PROGRAM Datalogger
VAR_IN_OUT CONSTANT
	monitoring			: ST_System_Monitor;
END_VAR

VAR
	FB_Datalogger					:FB_Datalogger;
END_VAR
VAR CONSTANT
	MAXLREALTOSTRINGLENGTH			: UDINT := 30;	
	NUMBEROFCOLUMNS					: UDINT := 40;													// Total number of columns
	TOTALNUMBEROFROWS				: UDINT := 86400;										    	// Total number of rows in one file (Depends of logtime)
	INCREOFROWS						: UDINT := 5;													// Amount of rows to write at once
	BUFFERMEM						: UDINT := 150;													// Effects file size
	NUMBEROFELEMENTS				: UDINT := NUMBEROFCOLUMNS * INCREOFROWS;						// > NUMBEROFCOLUMNS * INCREOFROWS
	MARGEDATAUSAGE					: REAL  := 0.05;												// 5% Standard marge (95% of storage gets used)
END_VAR
VAR PERSISTENT
	//Datalog presis 
	udi_MaxAmoutOfFiles									: UDINT;								// Max amount of files (30Mb = 12000 ROWS = 10min log)
	udi_AmountOfFiles									: UDINT;
	b_FileNotClosed										: BOOL;
	ui_FileNotClosed									: UINT; 
	a_LogFilesCreated									: ARRAY [0..10000] OF STRING(30);
END_VAR

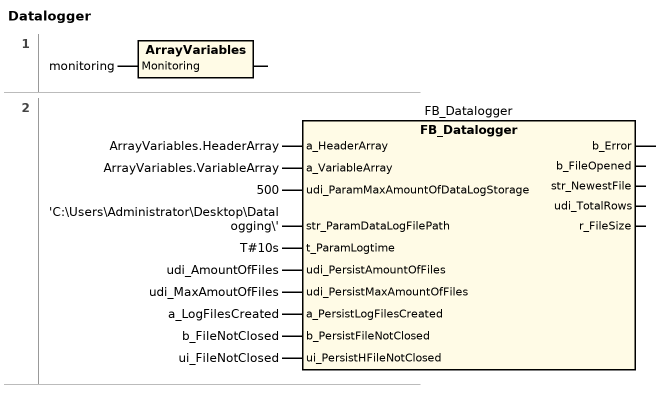
// NETWORK 1
ArrayVariables(Monitoring := monitoring);

// NETWORK 2
FB_Datalogger(
    a_HeaderArray := ArrayVariables.HeaderArray,
    a_VariableArray := ArrayVariables.VariableArray,
    udi_ParamMaxAmountOfDataLogStorage := 500,
    str_ParamDataLogFilePath := 'C:\Users\Administrator\Desktop\Datalogging\',
    t_ParamLogtime := T#10s,
    udi_PersistAmountOfFiles := udi_AmountOfFiles,
    udi_PersistMaxAmountOfFiles := udi_MaxAmoutOfFiles,
    a_PersistLogFilesCreated := a_LogFilesCreated,
    b_PersistFileNotClosed := b_FileNotClosed,
    ui_PersistHFileNotClosed := ui_FileNotClosed);

END_PROGRAM

(* stored: Version 1.1.0.1, ProductVersion 3.1.4024.12
   POU Datalogger: Id {9f3760cc-df04-417c-bc8e-220883b00970}, SpecialFunc None *)
